// TIA Portal project "SCDW_TEST_06997c36" (V17)

(* hardware
DEVICE "SCDW_FANGAS_PLC"  S7-1200 Station
   slot 0: "Rack_0"  S7-1200 Rack  Rack  V1.0
   slot 1: "SCDW_FANGAS_PLC"  CPU 1214C AC/DC/Rly  6ES7 214-1BG40-0XB0  V4.4
*)

// ===== PLC "SCDW_FANGAS_PLC"  CPU 1214C AC/DC/Rly =====

VAR_GLOBAL   // PLC tag table "SCDW_FANGAS_TAGS"
   "风机运行" AT %Q4.4 : Bool;
   "烧嘴电源" AT %Q4.6 : Bool;
   "风机控制" AT %QW44 : Int;
END_VAR

DATA_BLOCK "信号数据"   // DB1
{ S7_Optimized_Access := 'TRUE' }
VERSION : 0.1
   VAR
      风机运行按 : Bool;
      风机故障反馈 : Bool;
      风机手动 : Bool;
      风机自动输出 : Real;
      风机手动频率 : Real;
      风机控制输出 : Real;
      风压测量值 : Real;
   END_VAR
BEGIN
END_DATA_BLOCK

DATA_BLOCK "内部数据"   // DB2
{ S7_Optimized_Access := 'TRUE' }
VERSION : 0.1
   VAR
      风机控制输出值 : Real;
      风压过渡 : Int;
   END_VAR
BEGIN
END_DATA_BLOCK

FUNCTION "风机燃气_蓝图回归" : Void   // FC1, LAD
{ S7_Optimized_Access := 'TRUE' }
BEGIN

REGION Network 1: 程序段 1
   // 风机输出。将 %DB3.DBX129.4“信号数据”.“风机运行按”作为常开触点，与 %DB3.DBX129.4“信号数据”.“风机故障反馈”作为常闭触点串联，当风机运行按接通且风机故障反馈未动作时，驱动 %Q4.4“风机运行”线圈。随后建立风机自动/手动输出逻辑，以 %DB3.DBX129.3“信号数据”.“风机手动”作为模式选择信号。当“风机手动”为 FALSE 时，执行 MOVE 指令，将 %DB3.DBD130“信号数据”.“风机自动输出”的值直接赋给 %DB3.DBD138“信号数据”.“风机控制输出”；当“风机手动”为 TRUE 时，执行 MUL（REAL）指令，以 %DB3.DBD134“信号数据”.“风机手动频率”为 IN1、常数 2.0 为 IN2，相乘后的结果输出至 %DB3.DBD138“信号数据”.“风机控制输出”，即风机控制输出等于风机手动频率乘以 2.0
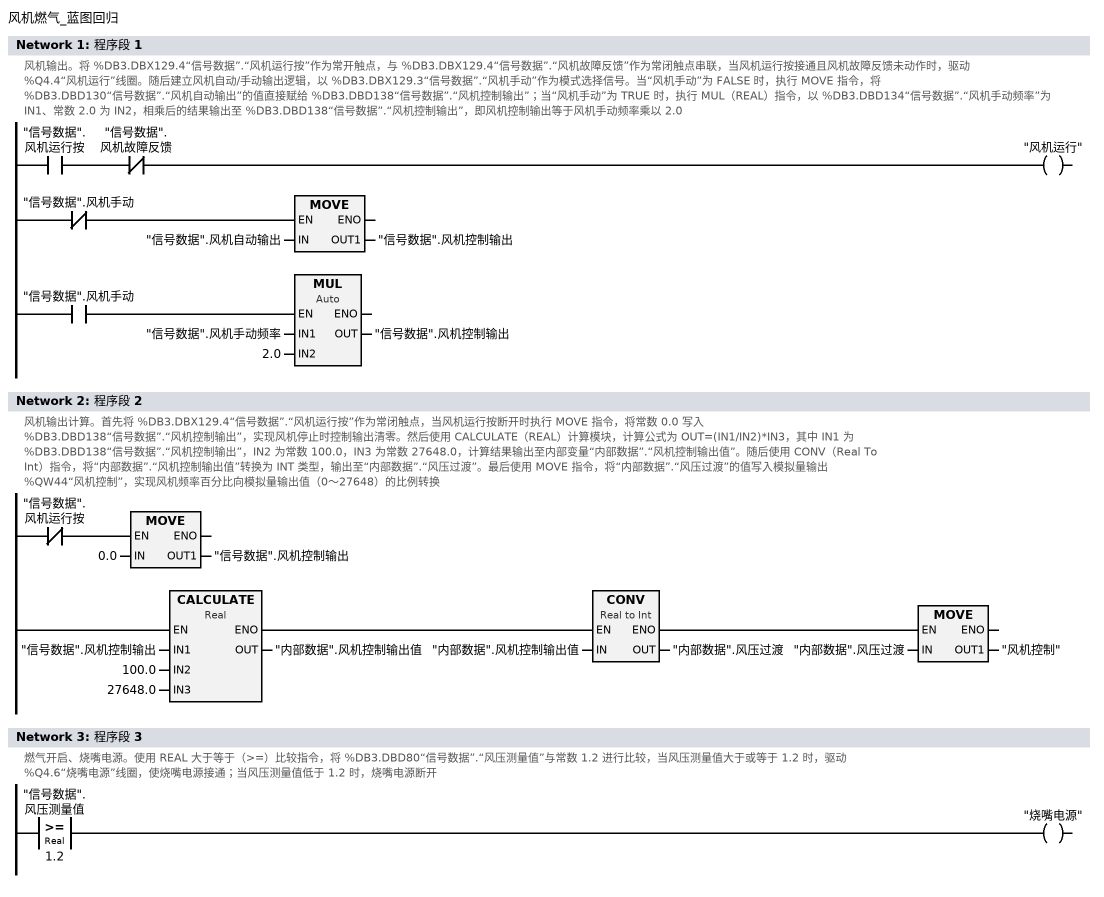
   RUNG wire#powerrail
      Contact( "信号数据".风机运行按 )
      I_Contact( "信号数据".风机故障反馈 )
      Coil( "风机运行" )
   END_RUNG
   RUNG wire#powerrail
      I_Contact( "信号数据".风机手动 )
      Move(in := "信号数据".风机自动输出, out1 => "信号数据".风机控制输出)
   END_RUNG
   RUNG wire#powerrail
      Contact( "信号数据".风机手动 )
      Mul(in1 := "信号数据".风机手动频率, in2 := 2.0, out => "信号数据".风机控制输出)
   END_RUNG
   // the same network as SCL:
   "风机运行" := "信号数据".风机运行按 AND NOT "信号数据".风机故障反馈;
   IF NOT "信号数据".风机手动 THEN "信号数据".风机控制输出 := "信号数据".风机自动输出; END_IF;
   IF "信号数据".风机手动 THEN "信号数据".风机控制输出 := "信号数据".风机手动频率 * 2.0; END_IF;
END_REGION

REGION Network 2: 程序段 2
   // 风机输出计算。首先将 %DB3.DBX129.4“信号数据”.“风机运行按”作为常闭触点，当风机运行按断开时执行 MOVE 指令，将常数 0.0 写入 %DB3.DBD138“信号数据”.“风机控制输出”，实现风机停止时控制输出清零。然后使用 CALCULATE（REAL）计算模块，计算公式为 OUT=(IN1/IN2)*IN3，其中 IN1 为 %DB3.DBD138“信号数据”.“风机控制输出”，IN2 为常数 100.0，IN3 为常数 27648.0，计算结果输出至内部变量“内部数据”.“风机控制输出值”。随后使用 CONV（Real To Int）指令，将“内部数据”.“风机控制输出值”转换为 INT 类型，输出至“内部数据”.“风压过渡”。最后使用 MOVE 指令，将“内部数据”.“风压过渡”的值写入模拟量输出 %QW44“风机控制”，实现风机频率百分比向模拟量输出值（0～27648）的比例转换
   RUNG wire#powerrail
      I_Contact( "信号数据".风机运行按 )
      Move(in := 0.0, out1 => "信号数据".风机控制输出)
   END_RUNG
   RUNG wire#powerrail
      { S7_Templates := "SrcType := Real"; S7_Expression := "(IN1/IN2)*IN3" } Calculate(in1 := "信号数据".风机控制输出, in2 := 100.0, in3 := 27648.0, out => "内部数据".风机控制输出值)
      { S7_Templates := "[SrcType := Real, DestType := Int]" } Convert(in := "内部数据".风机控制输出值, out => "内部数据".风压过渡)
      Move(in := "内部数据".风压过渡, out1 => "风机控制")
   END_RUNG
   // the same network as SCL:
   IF NOT "信号数据".风机运行按 THEN "信号数据".风机控制输出 := 0.0; END_IF;
   "内部数据".风机控制输出值 := ("信号数据".风机控制输出/100.0)*27648.0;
   "内部数据".风压过渡 := REAL_TO_INT("内部数据".风机控制输出值);
   "风机控制" := "内部数据".风压过渡;
END_REGION

REGION Network 3: 程序段 3
   // 燃气开启、烧嘴电源。使用 REAL 大于等于（>=）比较指令，将 %DB3.DBD80“信号数据”.“风压测量值”与常数 1.2 进行比较，当风压测量值大于或等于 1.2 时，驱动 %Q4.6“烧嘴电源”线圈，使烧嘴电源接通；当风压测量值低于 1.2 时，烧嘴电源断开
   RUNG wire#powerrail
      { S7_Templates := "SrcType := Real" } GE_Contact(in1 := "信号数据".风压测量值, in2 := 1.2)
      Coil( "烧嘴电源" )
   END_RUNG
   // the same network as SCL:
   "烧嘴电源" := "信号数据".风压测量值 >= 1.2;
END_REGION
END_FUNCTION

ORGANIZATION_BLOCK "Main"   // OB1, LAD, ProgramCycle
TITLE = "Main Program Sweep (Cycle)"
{ S7_Optimized_Access := 'TRUE' }
VERSION : 0.1
   VAR_INPUT
      Initial_Call : Bool;   // Initial call of this OB
      Remanence : Bool;   // =True, if remanent data are available
   END_VAR
BEGIN
END_ORGANIZATION_BLOCK